FUNCTION_BLOCK TEST_SUB (* Test SUB functions *)
  (* Standard: IEC 61499-1 *)
  (* Version 0.0, 2006-09-11, JHC, Holobloc Inc *)
  (* Compiler header: package fb.rt.test; *)
  (* Compiler classdef: SimpleFB *)
  (* Compiler Java Sun JDK 1.5.0 *)
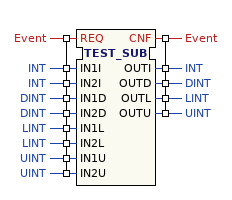
  EVENT_INPUT
    REQ WITH IN1I, IN2I, IN2D, IN1L, IN2L, IN1U, IN2U, IN1D;
  END_EVENT
  EVENT_OUTPUT
    CNF WITH OUTI, OUTD, OUTL, OUTU;
  END_EVENT
  VAR_INPUT
    IN1I : INT;
    IN2I : INT;
    IN1D : DINT;
    IN2D : DINT;
    IN1L : LINT;
    IN2L : LINT;
    IN1U : UINT;
    IN2U : UINT;
  END_VAR
  VAR_OUTPUT
    OUTI : INT;
    OUTD : DINT;
    OUTL : LINT;
    OUTU : UINT;
  END_VAR
  ALGORITHM REQ IN FBD:
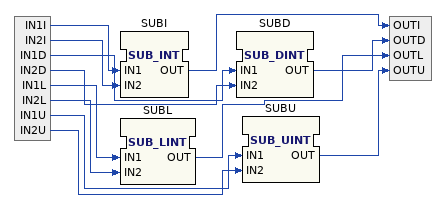
    FBS
      SUBI : SUB_INT;
      SUBD : SUB_DINT;
      SUBL : SUB_LINT;
      SUBU : SUB_UINT;
    END_FBS
    DATA_CONNECTIONS
      IN1I TO SUBI.IN1;
      IN2I TO SUBI.IN2;
      SUBI.OUT TO OUTI;
      IN1D TO SUBD.IN1;
      IN2D TO SUBD.IN2;
      SUBD.OUT TO OUTD;
      IN1L TO SUBL.IN1;
      IN2L TO SUBL.IN2;
      SUBL.OUT TO OUTL;
      IN1U TO SUBU.IN1;
      IN2U TO SUBU.IN2;
      SUBU.OUT TO OUTU;
    END_CONNECTIONS
  END_ALGORITHM
END_FUNCTION_BLOCK
